Fanuc KAREL source: kt00567.KL

PROGRAM KT00567
%STACKSIZE=65535
%PRIORITY=65535
%NOLOCKGROUP
VAR
R2 : REAL
-- UNRESOLVED DECLARATIONS (source type spelling not recovered)
-- V1 : TYPE_0x0013 (type_u16=0x0013)
-- OUT : TYPE_0x0013 (type_u16=0x0013)
BEGIN
-- UNSAFE_SOURCE_IR line 8: field_offset(V1,0) = 1065353216
R2=3.0
-- UNRESOLVED_PC line 10 opcodes [49 21 8A 4A] marker_code=36
END KT00567
